(* IEC 61131-3 sources: xPLCCore/codesys_code/Application (part 2) *)

(* ---- PRG_DiagReply.st ---- *)
PROGRAM PRG_DiagReply
VAR_INPUT
    // Request: one SYS packet copied in by TCP_MSGPAK_Server (Comm task),
    // ReqLen > 0 means "answer it this call"; cleared when done. Inputs,
    // so the caller may write them.
    ReqBuf  : ARRAY[0..255] OF BYTE;
    ReqLen  : UDINT;
END_VAR
VAR
    // Reply, ready for fbMyServer.Send when OutLen > 0 (one call = one reply).
    OutBuf  : ARRAY[0..2047] OF BYTE;
    OutLen  : UDINT;
    DiagInfo  : MsgPakInfo;
    xInfoInit : BOOL;

    // Same names as in AxisGroupSM so the handler code moved here on
    // 2026-10-05 reads unchanged (own instances: this is another task).
    MessagePackerFb       : FB_MpPacker;
    MessageUnpackerFb     : FB_MpUnpacker;
    ResponsePacketPointer : POINTER TO MsgPakInfo;
    CommandId   : DINT;
    CommandType : STRING;
    CommandAck  : BOOL;
    ShouldReturn : BOOL;

    HandledCount : UDINT;     // replies built
    UnknownCount : UDINT;     // a command routed here without a handler

    // Scratch (was AxisGroupSM.DrainHostPackets VAR).
    EcTrStr : STRING(255);    // EC_STATS trl / trh
    EcSnapK : INT;
    EcObjJ  : INT;
    EcObjKey : STRING(7);
    EcTrI   : INT;
    EcEvtFrom : UDINT;
    EcEvtI  : UDINT;
    // TASK_STATS scratch.
    TsH     : __XWORD;        // RTS_IEC_HANDLE
    TsR     : UDINT;          // RTS_IEC_RESULT, 0 = ERR_OK
    TsP     : POINTER TO CmpIecTask.Task_Info2;
    TsN     : INT;
    TsReset : BOOL;
    TsKey   : STRING(31);
    TsName  : STRING(63);
END_VAR
(* =========== IMPLEMENTATION =========== *)
// Read-only diagnostics answered in the Comm task (2026-10-05). These
// commands only read GVL / AxisGroupSM state (a few set a reset flag that
// the EtherCAT task consumes), and their replies are long (EC_STATS ~1 KB,
// TASK_STATS, DEM_STATS snap): built in the 1 ms EtherCAT task they could
// make a scan overrun. TCP_MSGPAK_Server copies the packet into ReqBuf and
// calls this program, then sends OutBuf itself, so the reply ring
// (reMP_info) keeps its single producer. Not in a task of its own.
//
// The handler bodies are the ones that lived in AxisGroupSM.DrainHostPackets;
// AxisGroupSM.* reads are a torn-read risk only in theory (diagnostics).
OutLen := 0;
IF ReqLen = 0 THEN
    RETURN;
END_IF;
IF NOT xInfoInit THEN
    DiagInfo := MsgPakInfoInit(ADR(OutBuf), 2048, TRUE);
    xInfoInit := TRUE;
END_IF;
MsgPakInfoClear(DiagInfo);
ResponsePacketPointer := ADR(DiagInfo);
MessagePackerFb.BindSlot(ResponsePacketPointer);
MessageUnpackerFb.Init(ADR(ReqBuf), ReqLen);
CommandId   := TO_DINT(MessageUnpackerFb.TryReadINT64('id', 0));
CommandType := MessageUnpackerFb.TryReadString('cmd', '');
CommandAck  := FALSE;
ShouldReturn := FALSE;

    IF (CommandType = 'SETTLE_TRACE') THEN
        // The last stop trace (GVL.Tr*): seq, at (PLC ms of the stop),
        // ev = up to 4 samples from index from:i (0..399, 100 = the
        // stop) as cx:cy:cz:ax:ay:az (mm), comma separated.
        ShouldReturn := TRUE;
        CommandAck := TRUE;
        ResponsePacketPointer^.ele_count := 0;
        EcTrI := LIMIT(0, LINT_TO_INT(MessageUnpackerFb.TryReadINT64('from', 0)), 399);
        MessagePackerFb.PackKvLint(ADR('seq'), UDINT_TO_LINT(GVL.TrSeq));
        MessagePackerFb.PackKvLint(ADR('at'), UDINT_TO_LINT(GVL.TrAtMs));
        EcTrStr := '';
        FOR EcObjJ := EcTrI TO MIN(EcTrI + 3, 399) DO
            EcTrStr := CONCAT(EcTrStr, REAL_TO_STRING(GVL.TrCX[EcObjJ]));
            EcTrStr := CONCAT(EcTrStr, ':');
            EcTrStr := CONCAT(EcTrStr, REAL_TO_STRING(GVL.TrCY[EcObjJ]));
            EcTrStr := CONCAT(EcTrStr, ':');
            EcTrStr := CONCAT(EcTrStr, REAL_TO_STRING(GVL.TrCZ[EcObjJ]));
            EcTrStr := CONCAT(EcTrStr, ':');
            EcTrStr := CONCAT(EcTrStr, REAL_TO_STRING(GVL.TrAX[EcObjJ]));
            EcTrStr := CONCAT(EcTrStr, ':');
            EcTrStr := CONCAT(EcTrStr, REAL_TO_STRING(GVL.TrAY[EcObjJ]));
            EcTrStr := CONCAT(EcTrStr, ':');
            EcTrStr := CONCAT(EcTrStr, REAL_TO_STRING(GVL.TrAZ[EcObjJ]));
            EcTrStr := CONCAT(EcTrStr, ',');
        END_FOR;
        MessagePackerFb.PackKvStr(ADR('ev'), ADR(EcTrStr));
    ELSIF (CommandType = 'SETTLE') THEN
        // Settling-time log (GVL.Settle*): n = stops so far, tol =
        // tolerance mm, ev = up to 20 stops from index from:i as
        // at_ms:settle_ms:err_at_stop_um. reset:1 clears it.
        ShouldReturn := TRUE;
        CommandAck := TRUE;
        ResponsePacketPointer^.ele_count := 0;
        IF MessageUnpackerFb.TryReadINT64('reset', 0) <> 0 THEN
            GVL.SettleN := 0;
        END_IF;
        EcEvtFrom := LINT_TO_UDINT(MessageUnpackerFb.TryReadINT64('from', 0));
        MessagePackerFb.PackKvLint(ADR('n'), UDINT_TO_LINT(GVL.SettleN));
        MessagePackerFb.PackKvReal(ADR('tol'), LREAL_TO_REAL(GVL.SettleTolMm));
        EcTrStr := '';
        EcEvtI := EcEvtFrom;
        WHILE (EcEvtI < GVL.SettleN) AND (EcEvtI < EcEvtFrom + 20) DO
            EcTrStr := CONCAT(EcTrStr, UDINT_TO_STRING(GVL.SettleAtMs[EcEvtI MOD 256]));
            EcTrStr := CONCAT(EcTrStr, ':');
            EcTrStr := CONCAT(EcTrStr, UDINT_TO_STRING(GVL.SettleMs[EcEvtI MOD 256]));
            EcTrStr := CONCAT(EcTrStr, ':');
            EcTrStr := CONCAT(EcTrStr, UDINT_TO_STRING(GVL.SettleErrUm[EcEvtI MOD 256]));
            EcTrStr := CONCAT(EcTrStr, ',');
            EcEvtI := EcEvtI + 1;
        END_WHILE;
        MessagePackerFb.PackKvStr(ADR('ev'), ADR(EcTrStr));
    ELSIF (CommandType = 'DWELL') THEN
        // Every-stop log (GVL.Dw*): n = stops so far, tol mm, hist =
        // settle time histogram (edges 1 2 5 10 15 20 50 ms, last =
        // not settled), emax = max error when leaving (um), ev = up
        // to 8 stops from index from:i as at_ms:dwell_ms:settle_ms:
        // err_stop_um:err_leave_um:err_5ms_um:err_10ms_um (settle 4294967295
        // = not settled; fields 6 and 7 since 2026-10-05); evq = the same
        // stops as buf:hostq:cool_ms:z_um (GVL.DwBuf / DwHostQ / DwCoolMs /
        // DwZUm, 2026-10-05; a separate string so ev stays within 255).
        // reset:1 clears it.
        ShouldReturn := TRUE;
        CommandAck := TRUE;
        ResponsePacketPointer^.ele_count := 0;
        IF MessageUnpackerFb.TryReadINT64('reset', 0) <> 0 THEN
            GVL.DwN := 0;
            GVL.DwErrLeaveMaxUm := 0;
            FOR EcObjJ := 0 TO 8 DO
                GVL.DwHist[EcObjJ] := 0;
            END_FOR;
        END_IF;
        EcEvtFrom := LINT_TO_UDINT(MessageUnpackerFb.TryReadINT64('from', 0));
        MessagePackerFb.PackKvLint(ADR('n'), UDINT_TO_LINT(GVL.DwN));
        MessagePackerFb.PackKvReal(ADR('tol'), LREAL_TO_REAL(GVL.SettleTolMm));
        MessagePackerFb.PackKvLint(ADR('emax'), UDINT_TO_LINT(GVL.DwErrLeaveMaxUm));
        EcTrStr := '';
        FOR EcObjJ := 0 TO 8 DO
            EcTrStr := CONCAT(EcTrStr, UDINT_TO_STRING(GVL.DwHist[EcObjJ]));
            EcTrStr := CONCAT(EcTrStr, ',');
        END_FOR;
        MessagePackerFb.PackKvStr(ADR('hist'), ADR(EcTrStr));
        EcTrStr := '';
        EcEvtI := EcEvtFrom;
        WHILE (EcEvtI < GVL.DwN) AND (EcEvtI < EcEvtFrom + 8) DO
            EcTrStr := CONCAT(EcTrStr, UDINT_TO_STRING(GVL.DwAtMs[EcEvtI MOD 4096]));
            EcTrStr := CONCAT(EcTrStr, ':');
            EcTrStr := CONCAT(EcTrStr, UDINT_TO_STRING(GVL.DwDwellMs[EcEvtI MOD 4096]));
            EcTrStr := CONCAT(EcTrStr, ':');
            EcTrStr := CONCAT(EcTrStr, UDINT_TO_STRING(GVL.DwSettleMs[EcEvtI MOD 4096]));
            EcTrStr := CONCAT(EcTrStr, ':');
            EcTrStr := CONCAT(EcTrStr, UDINT_TO_STRING(GVL.DwErr0Um[EcEvtI MOD 4096]));
            EcTrStr := CONCAT(EcTrStr, ':');
            EcTrStr := CONCAT(EcTrStr, UDINT_TO_STRING(GVL.DwErrLeaveUm[EcEvtI MOD 4096]));
            EcTrStr := CONCAT(EcTrStr, ':');
            EcTrStr := CONCAT(EcTrStr, UDINT_TO_STRING(GVL.DwErr5Um[EcEvtI MOD 4096]));
            EcTrStr := CONCAT(EcTrStr, ':');
            EcTrStr := CONCAT(EcTrStr, UDINT_TO_STRING(GVL.DwErr10Um[EcEvtI MOD 4096]));
            EcTrStr := CONCAT(EcTrStr, ',');
            EcEvtI := EcEvtI + 1;
        END_WHILE;
        MessagePackerFb.PackKvStr(ADR('ev'), ADR(EcTrStr));
        EcTrStr := '';
        EcEvtI := EcEvtFrom;
        WHILE (EcEvtI < GVL.DwN) AND (EcEvtI < EcEvtFrom + 8) DO
            EcTrStr := CONCAT(EcTrStr, UINT_TO_STRING(GVL.DwBuf[EcEvtI MOD 4096]));
            EcTrStr := CONCAT(EcTrStr, ':');
            EcTrStr := CONCAT(EcTrStr, UINT_TO_STRING(GVL.DwHostQ[EcEvtI MOD 4096]));
            EcTrStr := CONCAT(EcTrStr, ':');
            EcTrStr := CONCAT(EcTrStr, INT_TO_STRING(GVL.DwCoolMs[EcEvtI MOD 4096]));
            EcTrStr := CONCAT(EcTrStr, ':');
            EcTrStr := CONCAT(EcTrStr, DINT_TO_STRING(GVL.DwZUm[EcEvtI MOD 4096]));
            EcTrStr := CONCAT(EcTrStr, ',');
            EcEvtI := EcEvtI + 1;
        END_WHILE;
        MessagePackerFb.PackKvStr(ADR('evq'), ADR(EcTrStr));
    ELSIF (CommandType = 'FB_STATS') THEN
        // Feedback shock monitor (GVL.Fb*): per drive k, fd{k} =
        // histogram of |d2 actual position| (edges 1k 2k 5k 10k 20k
        // 50k 100k PUU), fdm{k} its max, ft{k} = histogram of |torque
        // change| (edges 5 10 20 50 100 200 500, 0.1 %), ftm{k} its
        // max, tq{k} = the torque now. reset:1 clears after the reply.
        ShouldReturn := TRUE;
        CommandAck := TRUE;
        ResponsePacketPointer^.ele_count := 0;
        FOR EcTrI := 0 TO 2 DO
            EcTrStr := '';
            FOR EcObjJ := 0 TO 7 DO
                EcTrStr := CONCAT(EcTrStr, UDINT_TO_STRING(GVL.FbD2Hist[EcTrI, EcObjJ]));
                EcTrStr := CONCAT(EcTrStr, ',');
            END_FOR;
            EcObjKey := CONCAT('fd', INT_TO_STRING(EcTrI));
            MessagePackerFb.PackKvStr(ADR(EcObjKey), ADR(EcTrStr));
            EcObjKey := CONCAT('fdm', INT_TO_STRING(EcTrI));
            MessagePackerFb.PackKvDint(ADR(EcObjKey), GVL.FbD2Max[EcTrI]);
            EcTrStr := '';
            FOR EcObjJ := 0 TO 7 DO
                EcTrStr := CONCAT(EcTrStr, UDINT_TO_STRING(GVL.FbTqHist[EcTrI, EcObjJ]));
                EcTrStr := CONCAT(EcTrStr, ',');
            END_FOR;
            EcObjKey := CONCAT('ft', INT_TO_STRING(EcTrI));
            MessagePackerFb.PackKvStr(ADR(EcObjKey), ADR(EcTrStr));
            EcObjKey := CONCAT('ftm', INT_TO_STRING(EcTrI));
            MessagePackerFb.PackKvDint(ADR(EcObjKey), INT_TO_DINT(GVL.FbTqMax[EcTrI]));
        END_FOR;
        MessagePackerFb.PackKvDint(ADR('tq0'), INT_TO_DINT(GVL.TorqueTap0));
        MessagePackerFb.PackKvDint(ADR('tq1'), INT_TO_DINT(GVL.TorqueTap1));
        MessagePackerFb.PackKvDint(ADR('tq2'), INT_TO_DINT(GVL.TorqueTap2));
        IF MessageUnpackerFb.TryReadINT64('reset', 0) <> 0 THEN
            GVL.FbReset := TRUE;
        END_IF;
    ELSIF (CommandType = 'ESP_SYNC') THEN
        // The EasyCAT SYNC0-interval log (GVL.SyncLog*): n = buckets
        // so far, now = the last deviation (ns), ev = up to 12
        // buckets from index from:i as ms:min:max (ns).
        ShouldReturn := TRUE;
        CommandAck := TRUE;
        ResponsePacketPointer^.ele_count := 0;
        EcEvtFrom := LINT_TO_UDINT(MessageUnpackerFb.TryReadINT64('from', 0));
        MessagePackerFb.PackKvLint(ADR('n'), UDINT_TO_LINT(GVL.SyncLogN));
        MessagePackerFb.PackKvDint(ADR('now'), INT_TO_DINT(GVL.EspSyncDevNs));
        EcTrStr := '';
        EcEvtI := EcEvtFrom;
        WHILE (EcEvtI < GVL.SyncLogN) AND (EcEvtI < EcEvtFrom + 12) DO
            EcTrStr := CONCAT(EcTrStr, UDINT_TO_STRING(GVL.SyncLogMs[EcEvtI MOD 4096]));
            EcTrStr := CONCAT(EcTrStr, ':');
            EcTrStr := CONCAT(EcTrStr, INT_TO_STRING(GVL.SyncLogMin[EcEvtI MOD 4096]));
            EcTrStr := CONCAT(EcTrStr, ':');
            EcTrStr := CONCAT(EcTrStr, INT_TO_STRING(GVL.SyncLogMax[EcEvtI MOD 4096]));
            EcTrStr := CONCAT(EcTrStr, ',');
            EcEvtI := EcEvtI + 1;
        END_WHILE;
        MessagePackerFb.PackKvStr(ADR('ev'), ADR(EcTrStr));
    ELSIF (CommandType = 'ESP_ARR') THEN
        // The EasyCAT frame-arrival log (GVL.ArrLog*): n = buckets so
        // far, now = the last arrival (us), ev = up to 12 buckets from
        // index from:i as ms:min:max (us), comma separated.
        ShouldReturn := TRUE;
        CommandAck := TRUE;
        ResponsePacketPointer^.ele_count := 0;
        EcEvtFrom := LINT_TO_UDINT(MessageUnpackerFb.TryReadINT64('from', 0));
        MessagePackerFb.PackKvLint(ADR('n'), UDINT_TO_LINT(GVL.ArrLogN));
        MessagePackerFb.PackKvDint(ADR('now'), UINT_TO_DINT(GVL.EspArrUs));
        EcTrStr := '';
        EcEvtI := EcEvtFrom;
        WHILE (EcEvtI < GVL.ArrLogN) AND (EcEvtI < EcEvtFrom + 12) DO
            EcTrStr := CONCAT(EcTrStr, UDINT_TO_STRING(GVL.ArrLogMs[EcEvtI MOD 4096]));
            EcTrStr := CONCAT(EcTrStr, ':');
            EcTrStr := CONCAT(EcTrStr, UINT_TO_STRING(GVL.ArrLogMin[EcEvtI MOD 4096]));
            EcTrStr := CONCAT(EcTrStr, ':');
            EcTrStr := CONCAT(EcTrStr, UINT_TO_STRING(GVL.ArrLogMax[EcEvtI MOD 4096]));
            EcTrStr := CONCAT(EcTrStr, ',');
            EcEvtI := EcEvtI + 1;
        END_WHILE;
        MessagePackerFb.PackKvStr(ADR('ev'), ADR(EcTrStr));
    ELSIF (CommandType = 'DEM_EVT') THEN
        // The delay-change event log of drive axis:k (GVL.DemEvt):
        // n = events so far, ev = up to 20 entries from index from:i
        // (ms * 4 + code, comma separated). Entries older than
        // n - 1024 are overwritten.
        ShouldReturn := TRUE;
        CommandAck := TRUE;
        ResponsePacketPointer^.ele_count := 0;
        EcTrI := LIMIT(0, LINT_TO_INT(MessageUnpackerFb.TryReadINT64('axis', 0)), 2);
        EcEvtFrom := LINT_TO_UDINT(MessageUnpackerFb.TryReadINT64('from', 0));
        MessagePackerFb.PackKvLint(ADR('n'), UDINT_TO_LINT(GVL.DemEvtN[EcTrI]));
        EcTrStr := '';
        EcEvtI := EcEvtFrom;
        WHILE (EcEvtI < GVL.DemEvtN[EcTrI]) AND (EcEvtI < EcEvtFrom + 20) DO
            EcTrStr := CONCAT(EcTrStr, UDINT_TO_STRING(GVL.DemEvt[EcTrI, EcEvtI MOD 1024]));
            EcTrStr := CONCAT(EcTrStr, ',');
            EcEvtI := EcEvtI + 1;
        END_WHILE;
        MessagePackerFb.PackKvStr(ADR('ev'), ADR(EcTrStr));
    ELSIF (CommandType = 'DEM_STATS') THEN
        // The drives' position demand (0x6062) vs the targets we sent
        // (GVL.Dem*, PRG_EventLog). Per drive k: ds{k} stale, dlate{k}
        // one cycle behind the nominal lag, dgl{k} / dmx{k} d2 glitches /
        // max, dlt{k} PLC ms of the last stale, dl{k} the lag histogram
        // as text (lag 0..6, none). nsnap = snapshots taken; snap:i adds
        // snapshot i (s_axis, s_ms, s_why, s_t0 / s_t1 and s_d0 / s_d1 =
        // cycles 0-15 / 16-31 of target / demand). reset:1 clears.
        ShouldReturn := TRUE;
        CommandAck := TRUE;
        ResponsePacketPointer^.ele_count := 0;
        MessagePackerFb.PackKvDint(ADR('lagnom'), INT_TO_DINT(GVL.DemLagNominal));
        FOR EcTrI := 0 TO 2 DO
            EcObjKey := CONCAT('ds', INT_TO_STRING(EcTrI));
            MessagePackerFb.PackKvLint(ADR(EcObjKey), UDINT_TO_LINT(GVL.DemStale[EcTrI]));
            EcObjKey := CONCAT('dlate', INT_TO_STRING(EcTrI));
            MessagePackerFb.PackKvLint(ADR(EcObjKey), UDINT_TO_LINT(GVL.DemLate[EcTrI]));
            EcObjKey := CONCAT('dgl', INT_TO_STRING(EcTrI));
            MessagePackerFb.PackKvLint(ADR(EcObjKey), UDINT_TO_LINT(GVL.DemGlitch[EcTrI]));
            EcObjKey := CONCAT('dmx', INT_TO_STRING(EcTrI));
            MessagePackerFb.PackKvDint(ADR(EcObjKey), GVL.DemD2Max[EcTrI]);
            EcObjKey := CONCAT('dlt', INT_TO_STRING(EcTrI));
            MessagePackerFb.PackKvLint(ADR(EcObjKey), UDINT_TO_LINT(GVL.DemLastStaleMs[EcTrI]));
            EcTrStr := '';
            FOR EcObjJ := 0 TO 7 DO
                EcTrStr := CONCAT(EcTrStr, UDINT_TO_STRING(GVL.DemLag[EcTrI, EcObjJ]));
                EcTrStr := CONCAT(EcTrStr, ',');
            END_FOR;
            EcObjKey := CONCAT('dl', INT_TO_STRING(EcTrI));
            MessagePackerFb.PackKvStr(ADR(EcObjKey), ADR(EcTrStr));
        END_FOR;
        FOR EcTrI := 0 TO 2 DO
            EcObjKey := CONCAT('soff', INT_TO_STRING(EcTrI));
            MessagePackerFb.PackKvLint(ADR(EcObjKey), UDINT_TO_LINT(GVL.SyncOffCount[EcTrI]));
            EcObjKey := CONCAT('sofl', INT_TO_STRING(EcTrI));
            MessagePackerFb.PackKvLint(ADR(EcObjKey), UDINT_TO_LINT(GVL.SyncOffAndLate[EcTrI]));
            EcObjKey := CONCAT('stat', INT_TO_STRING(EcTrI));
            CASE EcTrI OF
                0: MessagePackerFb.PackKvDint(ADR(EcObjKey), WORD_TO_DINT(GVL.StatusTap0));
                1: MessagePackerFb.PackKvDint(ADR(EcObjKey), WORD_TO_DINT(GVL.StatusTap1));
            ELSE
                MessagePackerFb.PackKvDint(ADR(EcObjKey), WORD_TO_DINT(GVL.StatusTap2));
            END_CASE;
        END_FOR;
        MessagePackerFb.PackKvDint(ADR('nsnap'), INT_TO_DINT(GVL.DemSnapN));
        EcTrI := LINT_TO_INT(MessageUnpackerFb.TryReadINT64('snap', -1));
        IF (EcTrI >= 0) AND (EcTrI < GVL.DemSnapN) THEN
            MessagePackerFb.PackKvDint(ADR('s_axis'), INT_TO_DINT(GVL.DemSnapAxis[EcTrI]));
            MessagePackerFb.PackKvLint(ADR('s_ms'), UDINT_TO_LINT(GVL.DemSnapMs[EcTrI]));
            MessagePackerFb.PackKvDint(ADR('s_why'), INT_TO_DINT(GVL.DemSnapWhy[EcTrI]));
            EcTrStr := '';
            FOR EcSnapK := 0 TO 31 DO
                IF (GVL.DemSnapS[EcTrI, EcSnapK] AND 16#4000) <> 0 THEN
                    EcTrStr := CONCAT(EcTrStr, '1');
                ELSE
                    EcTrStr := CONCAT(EcTrStr, '0');
                END_IF;
            END_FOR;
            MessagePackerFb.PackKvStr(ADR('s_sync'), ADR(EcTrStr));
            FOR EcObjJ := 0 TO 3 DO
                EcTrStr := '';
                FOR EcSnapK := 0 TO 15 DO
                    IF EcObjJ < 2 THEN
                        EcTrStr := CONCAT(EcTrStr, DINT_TO_STRING(GVL.DemSnapT[EcTrI, (EcObjJ MOD 2) * 16 + EcSnapK]));
                    ELSE
                        EcTrStr := CONCAT(EcTrStr, DINT_TO_STRING(GVL.DemSnapD[EcTrI, (EcObjJ MOD 2) * 16 + EcSnapK]));
                    END_IF;
                    EcTrStr := CONCAT(EcTrStr, ',');
                END_FOR;
                CASE EcObjJ OF
                    0: EcObjKey := 's_t0';
                    1: EcObjKey := 's_t1';
                    2: EcObjKey := 's_d0';
                ELSE
                    EcObjKey := 's_d1';
                END_CASE;
                MessagePackerFb.PackKvStr(ADR(EcObjKey), ADR(EcTrStr));
            END_FOR;
        END_IF;
        IF MessageUnpackerFb.TryReadINT64('reset', 0) <> 0 THEN
            GVL.DemReset := TRUE;
        END_IF;
    ELSIF (CommandType = 'EC_STATS') THEN
        // EtherCAT health: the master's frame statistics (lost /
        // tx_err / rx_err, updated every 100 cycles) and the task
        // timing monitor (GVL.EcProf*: cycles, late100 / late500 =
        // periods over nominal + 100 / 500 us, pmin / pmax us,
        // h0..h5 = |period - nominal| < 20/50/100/200/500/>=500 us,
        // dc_out = cycles with DC out of sync, agsm_max us). reset:1
        // starts all of them over after this reply.
        ShouldReturn := TRUE;
        CommandAck := TRUE;
        ResponsePacketPointer^.ele_count := 0;
        MessagePackerFb.PackKvLint(ADR('lost'), UDINT_TO_LINT(GVL.EcLostFrames));
        MessagePackerFb.PackKvLint(ADR('tx_err'), UDINT_TO_LINT(GVL.EcTxErrors));
        MessagePackerFb.PackKvLint(ADR('rx_err'), UDINT_TO_LINT(GVL.EcRxErrors));
        MessagePackerFb.PackKvLint(ADR('cycles'), UDINT_TO_LINT(GVL.EcProfCycles));
        MessagePackerFb.PackKvLint(ADR('late100'), UDINT_TO_LINT(GVL.EcLate100));
        MessagePackerFb.PackKvLint(ADR('late500'), UDINT_TO_LINT(GVL.EcLate500));
        MessagePackerFb.PackKvReal(ADR('pmin'), LREAL_TO_REAL(GVL.EcPeriodUsMin));
        MessagePackerFb.PackKvReal(ADR('pmax'), LREAL_TO_REAL(GVL.EcPeriodUsMax));
        MessagePackerFb.PackKvLint(ADR('h0'), UDINT_TO_LINT(GVL.EcPeriodHist[0]));
        MessagePackerFb.PackKvLint(ADR('h1'), UDINT_TO_LINT(GVL.EcPeriodHist[1]));
        MessagePackerFb.PackKvLint(ADR('h2'), UDINT_TO_LINT(GVL.EcPeriodHist[2]));
        MessagePackerFb.PackKvLint(ADR('h3'), UDINT_TO_LINT(GVL.EcPeriodHist[3]));
        MessagePackerFb.PackKvLint(ADR('h4'), UDINT_TO_LINT(GVL.EcPeriodHist[4]));
        MessagePackerFb.PackKvLint(ADR('h5'), UDINT_TO_LINT(GVL.EcPeriodHist[5]));
        MessagePackerFb.PackKvLint(ADR('dc_out'), UDINT_TO_LINT(GVL.EcDcOutCycles));
        MessagePackerFb.PackKvReal(ADR('agsm_max'), LREAL_TO_REAL(GVL.EcAgsmUsMax));
        // g0..2 / gms0..2 / d2m0..2: set-position glitches of the
        // delta joints (count, PLC ms of the last, max |d2| deg/cycle^2)
        MessagePackerFb.PackKvLint(ADR('g0'), UDINT_TO_LINT(GVL.SetGlitchCount[0]));
        MessagePackerFb.PackKvLint(ADR('g1'), UDINT_TO_LINT(GVL.SetGlitchCount[1]));
        MessagePackerFb.PackKvLint(ADR('g2'), UDINT_TO_LINT(GVL.SetGlitchCount[2]));
        MessagePackerFb.PackKvLint(ADR('gms0'), UDINT_TO_LINT(GVL.SetGlitchLastMs[0]));
        MessagePackerFb.PackKvLint(ADR('gms1'), UDINT_TO_LINT(GVL.SetGlitchLastMs[1]));
        MessagePackerFb.PackKvLint(ADR('gms2'), UDINT_TO_LINT(GVL.SetGlitchLastMs[2]));
        MessagePackerFb.PackKvReal(ADR('d2m0'), LREAL_TO_REAL(GVL.SetD2Max[0]));
        MessagePackerFb.PackKvReal(ADR('d2m1'), LREAL_TO_REAL(GVL.SetD2Max[1]));
        MessagePackerFb.PackKvReal(ADR('d2m2'), LREAL_TO_REAL(GVL.SetD2Max[2]));
        // tic_max / tic0..9: where the task's IEC code ends in the
        // DC cycle (us, 100 us bins); sm0..2 / se0..2: the drives'
        // 0x1C32:0B SM-event missed / :20 sync error (-1 = SDO
        // failed, sdo_err)
        MessagePackerFb.PackKvReal(ADR('tic_max'), LREAL_TO_REAL(GVL.EcTicUsMax));
        MessagePackerFb.PackKvLint(ADR('tic0'), UDINT_TO_LINT(GVL.EcTicHist[0]));
        MessagePackerFb.PackKvLint(ADR('tic1'), UDINT_TO_LINT(GVL.EcTicHist[1]));
        MessagePackerFb.PackKvLint(ADR('tic2'), UDINT_TO_LINT(GVL.EcTicHist[2]));
        MessagePackerFb.PackKvLint(ADR('tic3'), UDINT_TO_LINT(GVL.EcTicHist[3]));
        MessagePackerFb.PackKvLint(ADR('tic4'), UDINT_TO_LINT(GVL.EcTicHist[4]));
        MessagePackerFb.PackKvLint(ADR('tic5'), UDINT_TO_LINT(GVL.EcTicHist[5]));
        MessagePackerFb.PackKvLint(ADR('tic6'), UDINT_TO_LINT(GVL.EcTicHist[6]));
        MessagePackerFb.PackKvLint(ADR('tic7'), UDINT_TO_LINT(GVL.EcTicHist[7]));
        MessagePackerFb.PackKvLint(ADR('tic8'), UDINT_TO_LINT(GVL.EcTicHist[8]));
        MessagePackerFb.PackKvLint(ADR('tic9'), UDINT_TO_LINT(GVL.EcTicHist[9]));
        MessagePackerFb.PackKvDint(ADR('sm0'), GVL.DrvSmMissed[0]);
        MessagePackerFb.PackKvDint(ADR('sm1'), GVL.DrvSmMissed[1]);
        MessagePackerFb.PackKvDint(ADR('sm2'), GVL.DrvSmMissed[2]);
        MessagePackerFb.PackKvDint(ADR('se0'), GVL.DrvSyncErr[0]);
        MessagePackerFb.PackKvDint(ADR('se1'), GVL.DrvSyncErr[1]);
        MessagePackerFb.PackKvDint(ADR('se2'), GVL.DrvSyncErr[2]);
        MessagePackerFb.PackKvDint(ADR('sdo_err'), GVL.EcSdoErr);
        MessagePackerFb.PackKvLint(ADR('bus_us'), DWORD_TO_LINT(AxisGroupSM.BusPeriodUs));   // EtherCAT_Task interval as read
        // Comm task profile: cs0..2 worst segment us (TCP server / MbProbe / EspHttp),
        // cb0..2 bus cycles inside it, co0..2 segments > 1 ms, cscan worst whole scan
        MessagePackerFb.PackKvReal(ADR('cs0'), LREAL_TO_REAL(GVL.CommSegUsMax[0]));
        MessagePackerFb.PackKvLint(ADR('cb0'), UDINT_TO_LINT(GVL.CommSegBusCyc[0]));
        MessagePackerFb.PackKvLint(ADR('co0'), UDINT_TO_LINT(GVL.CommSegOver1ms[0]));
        MessagePackerFb.PackKvReal(ADR('cs1'), LREAL_TO_REAL(GVL.CommSegUsMax[1]));
        MessagePackerFb.PackKvLint(ADR('cb1'), UDINT_TO_LINT(GVL.CommSegBusCyc[1]));
        MessagePackerFb.PackKvLint(ADR('co1'), UDINT_TO_LINT(GVL.CommSegOver1ms[1]));
        MessagePackerFb.PackKvReal(ADR('cs2'), LREAL_TO_REAL(GVL.CommSegUsMax[2]));
        MessagePackerFb.PackKvLint(ADR('cb2'), UDINT_TO_LINT(GVL.CommSegBusCyc[2]));
        MessagePackerFb.PackKvLint(ADR('co2'), UDINT_TO_LINT(GVL.CommSegOver1ms[2]));
        MessagePackerFb.PackKvReal(ADR('cscan'), LREAL_TO_REAL(GVL.CommScanUsMax));
        // fj0..3 / fm0..3 / fl0..3: following-error jumps (EAxis0..2, reel): count, max, PLC ms of the last
        MessagePackerFb.PackKvLint(ADR('fj0'), UDINT_TO_LINT(GVL.FeJumpCount[0]));
        MessagePackerFb.PackKvReal(ADR('fm0'), LREAL_TO_REAL(GVL.FeJumpMax[0]));
        MessagePackerFb.PackKvLint(ADR('fl0'), UDINT_TO_LINT(GVL.FeLastJumpMs[0]));
        MessagePackerFb.PackKvLint(ADR('fj1'), UDINT_TO_LINT(GVL.FeJumpCount[1]));
        MessagePackerFb.PackKvReal(ADR('fm1'), LREAL_TO_REAL(GVL.FeJumpMax[1]));
        MessagePackerFb.PackKvLint(ADR('fl1'), UDINT_TO_LINT(GVL.FeLastJumpMs[1]));
        MessagePackerFb.PackKvLint(ADR('fj2'), UDINT_TO_LINT(GVL.FeJumpCount[2]));
        MessagePackerFb.PackKvReal(ADR('fm2'), LREAL_TO_REAL(GVL.FeJumpMax[2]));
        MessagePackerFb.PackKvLint(ADR('fl2'), UDINT_TO_LINT(GVL.FeLastJumpMs[2]));
        MessagePackerFb.PackKvLint(ADR('fj3'), UDINT_TO_LINT(GVL.FeJumpCount[3]));
        MessagePackerFb.PackKvReal(ADR('fm3'), LREAL_TO_REAL(GVL.FeJumpMax[3]));
        MessagePackerFb.PackKvLint(ADR('fl3'), UDINT_TO_LINT(GVL.FeLastJumpMs[3]));
        MessagePackerFb.PackKvReal(ADR('ctask'), LREAL_TO_REAL(GVL.CommTaskUsMax));
        MessagePackerFb.PackKvReal(ADR('cout'), LREAL_TO_REAL(GVL.CommOutsideUsMax));
        MessagePackerFb.PackKvLint(ADR('cout500'), UDINT_TO_LINT(GVL.CommOutsideOver500));
        IF MessageUnpackerFb.TryReadINT64('obj', 0) <> 0 THEN  // long text: only on request
            // o0..o2: drive k's sync objects (DrvObj), "v,v,..." text
            FOR EcTrI := 0 TO 2 DO
                EcTrStr := '';
                FOR EcObjJ := 0 TO 11 DO
                    EcTrStr := CONCAT(EcTrStr, DINT_TO_STRING(GVL.DrvObj[EcTrI, EcObjJ]));
                    EcTrStr := CONCAT(EcTrStr, ',');
                END_FOR;
                EcObjKey := CONCAT('o', INT_TO_STRING(EcTrI));
                MessagePackerFb.PackKvStr(ADR(EcObjKey), ADR(EcTrStr));
            END_FOR;
        END_IF;
        // dg0..2 / dd0..2: the same glitch check on the integer
        // target sent to the drive (diSetPosition): count, max |d2|
        MessagePackerFb.PackKvLint(ADR('dg0'), UDINT_TO_LINT(GVL.DiGlitchCount[0]));
        MessagePackerFb.PackKvLint(ADR('dg1'), UDINT_TO_LINT(GVL.DiGlitchCount[1]));
        MessagePackerFb.PackKvLint(ADR('dg2'), UDINT_TO_LINT(GVL.DiGlitchCount[2]));
        MessagePackerFb.PackKvDint(ADR('dd0'), GVL.DiD2Max[0]);
        MessagePackerFb.PackKvDint(ADR('dd1'), GVL.DiD2Max[1]);
        MessagePackerFb.PackKvDint(ADR('dd2'), GVL.DiD2Max[2]);
        // tap*: the Target Position in the output image (read-only AT taps)
        MessagePackerFb.PackKvLint(ADR('tg0'), UDINT_TO_LINT(GVL.TapGlitch[0]));
        MessagePackerFb.PackKvDint(ADR('td0'), GVL.TapD2Max[0]);
        MessagePackerFb.PackKvLint(ADR('tnow0'), UDINT_TO_LINT(GVL.TapEqNow[0]));
        MessagePackerFb.PackKvLint(ADR('tprev0'), UDINT_TO_LINT(GVL.TapEqPrev[0]));
        MessagePackerFb.PackKvLint(ADR('tnone0'), UDINT_TO_LINT(GVL.TapEqNone[0]));
        MessagePackerFb.PackKvLint(ADR('tg1'), UDINT_TO_LINT(GVL.TapGlitch[1]));
        MessagePackerFb.PackKvDint(ADR('td1'), GVL.TapD2Max[1]);
        MessagePackerFb.PackKvLint(ADR('tnow1'), UDINT_TO_LINT(GVL.TapEqNow[1]));
        MessagePackerFb.PackKvLint(ADR('tprev1'), UDINT_TO_LINT(GVL.TapEqPrev[1]));
        MessagePackerFb.PackKvLint(ADR('tnone1'), UDINT_TO_LINT(GVL.TapEqNone[1]));
        MessagePackerFb.PackKvLint(ADR('tg2'), UDINT_TO_LINT(GVL.TapGlitch[2]));
        MessagePackerFb.PackKvDint(ADR('td2'), GVL.TapD2Max[2]);
        MessagePackerFb.PackKvLint(ADR('tnow2'), UDINT_TO_LINT(GVL.TapEqNow[2]));
        MessagePackerFb.PackKvLint(ADR('tprev2'), UDINT_TO_LINT(GVL.TapEqPrev[2]));
        MessagePackerFb.PackKvLint(ADR('tnone2'), UDINT_TO_LINT(GVL.TapEqNone[2]));
        // EasyCAT bus timing probe: e_stale / e_skip since reset,
        // e_late last second, e_late_sum since reset (the arrival
        // min / max moved to the per-100-ms ArrLog, SYS ESP_ARR)
        MessagePackerFb.PackKvDint(ADR('e_stale'), UINT_TO_DINT(GVL.EspStale - GVL.EspStale0));
        MessagePackerFb.PackKvDint(ADR('e_skip'), UINT_TO_DINT(GVL.EspSkip - GVL.EspSkip0));
        MessagePackerFb.PackKvDint(ADR('e_late'), UINT_TO_DINT(GVL.EspLate));
        MessagePackerFb.PackKvLint(ADR('e_late_sum'), UDINT_TO_LINT(GVL.EspLateSum));
        // e_pg / e_pd2 / e_pd2peak: EAxis0's target stream checked on the ESP32
        MessagePackerFb.PackKvDint(ADR('e_pg'), UINT_TO_DINT(GVL.EspPosGlitch - GVL.EspPosGlitch0));
        MessagePackerFb.PackKvLint(ADR('e_pd2'), UDINT_TO_LINT(GVL.EspPosD2Max));
        MessagePackerFb.PackKvLint(ADR('e_pd2peak'), UDINT_TO_LINT(GVL.EspPosD2Peak));
        IF MessageUnpackerFb.TryReadINT64('tr', 0) <> 0 THEN   // long text: only on request
            // trl / trh: the last 20 x 500 ms min / max of the above,
            // oldest first ("lo0,..." as text, us)
            EcTrStr := '';
            FOR EcTrI := 0 TO 19 DO
                EcTrStr := CONCAT(EcTrStr, REAL_TO_STRING(GVL.EcTicTrMin[(GVL.EcTicIdx + EcTrI) MOD 20]));
                EcTrStr := CONCAT(EcTrStr, ',');
            END_FOR;
            MessagePackerFb.PackKvStr(ADR('trl'), ADR(EcTrStr));
            EcTrStr := '';
            FOR EcTrI := 0 TO 19 DO
                EcTrStr := CONCAT(EcTrStr, REAL_TO_STRING(GVL.EcTicTrMax[(GVL.EcTicIdx + EcTrI) MOD 20]));
                EcTrStr := CONCAT(EcTrStr, ',');
            END_FOR;
            MessagePackerFb.PackKvStr(ADR('trh'), ADR(EcTrStr));
        END_IF;
        IF MessageUnpackerFb.TryReadINT64('reset', 0) <> 0 THEN
            GVL.EcProfReset := TRUE;
            GVL.EcStatsClear := TRUE;
            GVL.CommProfReset := TRUE;
        END_IF;
    ELSIF (CommandType = 'TASK_STATS') THEN
        // The runtime's task statistics -- what the IDE's Task
        // Configuration > Monitor shows -- for every task of the
        // application, SoftMotion's planning task included. Flat
        // keys per task k: tk_name, tk_prio, tk_interval_us,
        // tk_last / tk_avg / tk_max / tk_min (cycle time, us),
        // tk_jit / tk_jmin / tk_jmax (jitter, us), tk_cycles,
        // tk_iec_cycles; n = tasks. reset:true zeroes them after
        // reading (as the IDE's reset does).
        ShouldReturn := TRUE;
        CommandAck := TRUE;
        ResponsePacketPointer^.ele_count := 0;
        TsReset := MessageUnpackerFb.TryReadINT64('reset', 0) <> 0;
        TsN := 0;
        TsH := CmpIecTask.IecTaskGetFirst(ADR('Application'), ADR(TsR));
        WHILE (TsR = 0) AND (TsN < 8) DO
            TsP := CmpIecTask.IecTaskGetInfo3(TsH, ADR(TsR));
            IF TsP <> 0 THEN
                IF TsP^.pszName <> 0 THEN
                    TsName := TsP^.pszName^;
                ELSE
                    TsName := '?';
                END_IF;
                TsKey := CONCAT(CONCAT('t', INT_TO_STRING(TsN)), '_name');
                MessagePackerFb.PackKvStr(ADR(TsKey), ADR(TsName));
                TsKey := CONCAT(CONCAT('t', INT_TO_STRING(TsN)), '_prio');
                MessagePackerFb.PackKvDint(ADR(TsKey), TsP^.nPriority);
                TsKey := CONCAT(CONCAT('t', INT_TO_STRING(TsN)), '_interval_us');
                MessagePackerFb.PackKvLint(ADR(TsKey), DWORD_TO_LINT(TsP^.dwInterval));
                TsKey := CONCAT(CONCAT('t', INT_TO_STRING(TsN)), '_last');
                MessagePackerFb.PackKvLint(ADR(TsKey), DWORD_TO_LINT(TsP^.dwCycleTime));
                TsKey := CONCAT(CONCAT('t', INT_TO_STRING(TsN)), '_avg');
                MessagePackerFb.PackKvLint(ADR(TsKey), DWORD_TO_LINT(TsP^.dwAverageCycleTime));
                TsKey := CONCAT(CONCAT('t', INT_TO_STRING(TsN)), '_max');
                MessagePackerFb.PackKvLint(ADR(TsKey), DWORD_TO_LINT(TsP^.dwMaxCycleTime));
                TsKey := CONCAT(CONCAT('t', INT_TO_STRING(TsN)), '_min');
                MessagePackerFb.PackKvLint(ADR(TsKey), DWORD_TO_LINT(TsP^.dwMinCycleTime));
                TsKey := CONCAT(CONCAT('t', INT_TO_STRING(TsN)), '_jit');
                MessagePackerFb.PackKvDint(ADR(TsKey), TsP^.iJitter);
                TsKey := CONCAT(CONCAT('t', INT_TO_STRING(TsN)), '_jmin');
                MessagePackerFb.PackKvDint(ADR(TsKey), TsP^.iJitterMin);
                TsKey := CONCAT(CONCAT('t', INT_TO_STRING(TsN)), '_jmax');
                MessagePackerFb.PackKvDint(ADR(TsKey), TsP^.iJitterMax);
                TsKey := CONCAT(CONCAT('t', INT_TO_STRING(TsN)), '_cycles');
                MessagePackerFb.PackKvLint(ADR(TsKey), DWORD_TO_LINT(TsP^.dwCycleCount));
                TsKey := CONCAT(CONCAT('t', INT_TO_STRING(TsN)), '_iec_cycles');
                MessagePackerFb.PackKvLint(ADR(TsKey), DWORD_TO_LINT(TsP^.dwIECCycleCount));
                TsN := TsN + 1;
            END_IF;
            IF TsReset THEN
                CmpIecTask.IecTaskResetStatistics(TsH);
            END_IF;
            TsH := CmpIecTask.IecTaskGetNext(ADR('Application'), TsH, ADR(TsR));
        END_WHILE;
        MessagePackerFb.PackKvDint(ADR('n'), TsN);
    ELSIF (CommandType = 'VERSION') THEN
        // Build provenance: lets an external tool verify the running
        // PLC matches a repo commit without IDE assistance. Stamped by
        // codesys_scripts/jobs/stamp_build_info.py before import_all.
        ShouldReturn := TRUE;
        CommandAck := TRUE;
        ResponsePacketPointer^.ele_count := 0;
        MessagePackerFb.PackKvStr(ADR('git_sha'), ADR(GVL.BUILD_GIT_SHA));
        MessagePackerFb.PackKvLint(ADR('build_ts_ms'), GVL.BUILD_TS_MS);
        MessagePackerFb.PackKvLint(ADR('runtime_ms'), AxisGroupSM.RuntimeMs);
    ELSIF (CommandType = 'GET_DIAG') THEN
        // Generic comm/robustness counters dump. UI dashboard polls this
        // (e.g. once per second) to chart drop/NAK/reset rates and the
        // PING gap-jitter envelope. Read-only; doesn't perturb FSM.
        // Counters resettable via SYS/RESET_DBG_INFO (see existing handler).
        ShouldReturn := TRUE;
        CommandAck := TRUE;
        // GET_DIAG fields extended 2026-06-17 to be a TCP-side
        // superset of the daemon-side counter dump the fuzz tests
        // used to call via oapp.read_value. Lets fuzz/soak tests run
        // without the CODESYS RPC daemon being alive -- daemon dies
        // mid-test no longer breaks the test. New fields:
        //   self_reentry, pending_stchg_drop, pending_movedone_drop,
        //   remp_drop_reply, remp_drop_trig, dupe_cmd,
        //   io_cmd_count, io_trig_count, flyevent_avail
        ResponsePacketPointer^.ele_count := 0;
        MessagePackerFb.PackKvDint(ADR('remp_overflow_drop'), TO_DINT(GVL.ReMpOverflowDropCount));
        MessagePackerFb.PackKvLint(ADR('runtime_ms'), AxisGroupSM.RuntimeMs);
        MessagePackerFb.PackKvDint(ADR('sm_scans'), TO_DINT(GVL.AxisGroupSMScans));
        MessagePackerFb.PackKvDint(ADR('remp_drop'), TO_DINT(GVL.ReMpDropCount));
        MessagePackerFb.PackKvDint(ADR('overlen_drop'), TO_DINT(GVL.OverlenDropCount));
        MessagePackerFb.PackKvDint(ADR('send_stall_drop'), TO_DINT(GVL.SendStallDropCount));
        MessagePackerFb.PackKvDint(ADR('group_not_ready_nak'), TO_DINT(GVL.GroupNotReadyNakCount));
        MessagePackerFb.PackKvDint(ADR('missing_type_nak'), TO_DINT(GVL.MissingTypeFieldNakCount));
        MessagePackerFb.PackKvDint(ADR('coord_not_cfg_nak'), TO_DINT(GVL.CoordNotConfiguredNakCount));
        MessagePackerFb.PackKvDint(ADR('proto_mismatch_nak'), TO_DINT(GVL.ProtocolVersionMismatchCount));
        MessagePackerFb.PackKvDint(ADR('idle_reset'), TO_DINT(GVL.IdleResetCount));
        MessagePackerFb.PackKvDint(ADR('read_err_reset'), TO_DINT(GVL.ReadErrorResetCount));
        MessagePackerFb.PackKvDint(ADR('parser_err_reset'), TO_DINT(GVL.ParserErrorResetCount));
        MessagePackerFb.PackKvDint(ADR('write_err_reset'), TO_DINT(GVL.WriteErrorResetCount));
        MessagePackerFb.PackKvDint(ADR('client_connect_count'), TO_DINT(GVL.ClientConnectCount));
        MessagePackerFb.PackKvDint(ADR('server_long_idle_count'), TO_DINT(GVL.ServerLongIdleCount));
        MessagePackerFb.PackKvBool(ADR('server_active'), TCP_MSGPAK_Server.fbMyServer.xServerActive);
        MessagePackerFb.PackKvStr(ADR('bind_addr'), ADR(TCP_MSGPAK_Server.ipServerAddress.ipAddress));
        MessagePackerFb.PackKvDint(ADR('ui_ping_count'), TO_DINT(GVL.UiPingCount));
        MessagePackerFb.PackKvDint(ADR('ui_hb_stale_count'), TO_DINT(GVL.UiHeartbeatStaleCount));
        MessagePackerFb.PackKvDint(ADR('group_error_stop_trips'), TO_DINT(GVL.GroupErrorStopTripCount));
        MessagePackerFb.PackKvDint(ADR('ping_max_gap_ms'), TO_DINT(GVL.PingMaxGapMs));
        MessagePackerFb.PackKvLint(ADR('last_ui_ping_ms'), GVL.LastUiPingMs);
        MessagePackerFb.PackKvDint(ADR('st_chg_event_count'), TO_DINT(GVL.StateChangeEventCount));
        MessagePackerFb.PackKvDint(ADR('self_reentry'), TO_DINT(GVL.SelfReentryCount));
        MessagePackerFb.PackKvDint(ADR('pending_stchg_drop'), TO_DINT(GVL.PendingStChgDropCount));
        MessagePackerFb.PackKvDint(ADR('pending_movedone_drop'), TO_DINT(GVL.PendingMoveDoneDropCount));
        MessagePackerFb.PackKvDint(ADR('remp_drop_reply'), TO_DINT(GVL.ReMpDropCount_Reply));
        MessagePackerFb.PackKvDint(ADR('remp_drop_trig'), TO_DINT(GVL.ReMpDropCount_TriggerEvent));
        MessagePackerFb.PackKvDint(ADR('dupe_cmd'), TO_DINT(GVL.DupeCommandCount));
        // R2/R3/R4/R5/R11: new NAK counters. Published here => they
        // are part of the canonical ResetDiagCounters list (R8).
        MessagePackerFb.PackKvDint(ADR('unknown_cmd_nak'), TO_DINT(GVL.UnknownCmdNakCount));
        MessagePackerFb.PackKvDint(ADR('flyevent_reject_nak'), TO_DINT(GVL.FlyEventRejectNakCount));
        MessagePackerFb.PackKvDint(ADR('flyevent_full_nak'), TO_DINT(GVL.FlyEventBufferFullNakCount));
        MessagePackerFb.PackKvDint(ADR('io_cmd_count'), TO_DINT(AxisGroupSM.IoCommandCount));
        MessagePackerFb.PackKvDint(ADR('io_trig_count'), TO_DINT(AxisGroupSM.IoTriggerCount));
        MessagePackerFb.PackKvDint(ADR('flyevent_avail'), TO_DINT(AxisGroupSM.FlyEventAvailableCount));
ELSE
    CommandAck := FALSE;
    ResponsePacketPointer^.ele_count := 0;
    MessagePackerFb.PackKvStr(ADR('err'), ADR('unknown SYS cmd'));
    UnknownCount := UnknownCount + 1;
END_IF;

MessagePackerFb.PackKvDint(ADR('id'), CommandId);
MessagePackerFb.PackKvBool(ADR('ack'), CommandAck);
IF MsgPakInfoWrapup(DiagInfo) THEN
    OutLen := DiagInfo.buf_size;
    HandledCount := HandledCount + 1;
END_IF;
ReqLen := 0;

(* ---- PRG_EcatEsp.st ---- *)
PROGRAM PRG_EcatEsp
VAR
    byOut0          : USINT;        // bit 0 -> ESP32 LED
    byOut1          : USINT := 16#5A; // echoed back on in1
    byIn0           : USINT;        // ESP32 heartbeat counter
    byIn1           : USINT;        // echo of out1
    byLastIn0       : USINT;
    udiCounterSeen  : UDINT;        // cycles the heartbeat moved
    uiStaleCycles   : UINT;         // cycles since it last moved
    xEspAlive       : BOOL;         // heartbeat moved within 100 cycles
    xRoundTripOk    : BOOL;

    // QY2204-IIC (AS5600) encoder
    uiEncRaw        : UINT;         // 0..4095, one turn
    rEncDeg         : REAL;         // 0..360
    diEncPos        : DINT;         // multi-turn counts, from ESP32 power-up
    rEncTurns       : REAL;         // diEncPos / 4096
    byEncStatus     : USINT;        // bit5 MD, bit4 ML weak, bit3 MH strong, bit0 no sensor
    xMagnetOk       : BOOL;         // MD and neither too weak nor too strong
    xSensorMissing  : BOOL;
    byEncI2cErr     : USINT;
    byEncAgc        : USINT;
END_VAR
(* =========== IMPLEMENTATION =========== *)
GVL.EcProfT1 := LTIME();     // AxisGroupSM done (task timing monitor, PRG_EventLog)
ecat_esp_out0 := byOut0;
ecat_esp_out1 := byOut1;
byIn0 := ecat_esp_in0;
byIn1 := ecat_esp_in1;

IF byIn0 <> byLastIn0 THEN
    udiCounterSeen := udiCounterSeen + 1;
    uiStaleCycles := 0;
ELSIF uiStaleCycles < 65535 THEN
    uiStaleCycles := uiStaleCycles + 1;
END_IF
byLastIn0 := byIn0;
xEspAlive := uiStaleCycles < 100;
xRoundTripOk := (byIn1 = byOut1);

uiEncRaw := USINT_TO_UINT(ecat_esp_in2) OR SHL(USINT_TO_UINT(ecat_esp_in3), 8);
rEncDeg := UINT_TO_REAL(uiEncRaw) * 360.0 / 4096.0;
diEncPos := UDINT_TO_DINT(USINT_TO_UDINT(ecat_esp_in5)
                       OR SHL(USINT_TO_UDINT(ecat_esp_in6), 8)
                       OR SHL(USINT_TO_UDINT(ecat_esp_in7), 16)
                       OR SHL(USINT_TO_UDINT(ecat_esp_in8), 24));
rEncTurns := DINT_TO_REAL(diEncPos) / 4096.0;
byEncStatus := ecat_esp_in4;
xSensorMissing := (byEncStatus AND 16#01) <> 0;
xMagnetOk := ((byEncStatus AND 16#20) <> 0) AND ((byEncStatus AND 16#18) = 0) AND NOT xSensorMissing;
byEncI2cErr := ecat_esp_in9;
byEncAgc := ecat_esp_in10;

(* ---- PRG_EcatEspHttp.st ---- *)
PROGRAM PRG_EcatEspHttp
VAR CONSTANT
    HTML_LEN        : UDINT := 3061;
END_VAR
VAR
    iProfK          : INT;          // Comm task profile
    lrSegUs         : LREAL;
    sHtml           : STRING(3062) := '<!DOCTYPE html><html><head><meta charset="utf-8"><meta name="viewport" content="width=device-width,initial-scale=1"><title>EasyCAT &#32232;&#30908;&#22120;</title><style>body{font-family:system-ui,sans-serif;background:#f4f5f7;color:#1f2328;margin:0;padding:16px}h1{font-size:18px;margin:0 0 12px}.row{display:flex;flex-wrap:wrap;gap:12px}.card{background:#fff;border-radius:10px;padding:14px 16px;box-shadow:0 1px 3px rgba(0,0,0,.08);min-width:150px}.k{font-size:12px;color:#656d76}.v{font-size:26px;font-weight:600;font-variant-numeric:tabular-nums}.ok{color:#1a7f37}.bad{color:#cf222e}.warn{color:#9a6700}svg{display:block}#conn{font-size:12px;color:#656d76;margin-top:12px}</style></head><body><h1>EasyCAT + ESP32 &#32232;&#30908;&#22120;&#29376;&#24907;</h1><div class="row"><div class="card"><svg width="170" height="170" viewBox="-85 -85 170 170"><circle r="78" fill="#f4f5f7" stroke="#d0d7de" stroke-width="2"/><line id="nd" x1="0" y1="0" x2="0" y2="-68" stroke="#0969da" stroke-width="5" stroke-linecap="round"/><circle r="5" fill="#0969da"/></svg></div><div class="card"><div class="k">&#35282;&#24230;</div><div class="v" id="deg">-</div><div class="k" style="margin-top:10px">&#21407;&#22987;&#20540; (0-4095)</div><div class="v" id="raw">-</div></div><div class="card"><div class="k">&#22810;&#22280;&#20301;&#32622; (counts)</div><div class="v" id="pos">-</div><div class="k" style="margin-top:10px">&#22280;&#25976;</div><div class="v" id="turns">-</div></div></div><div class="row" style="margin-top:12px"><div class="card"><div class="k">ESP32</div><div class="v" id="alive">-</div></div><div class="card"><div class="k">EtherCAT</div><div class="v" id="ecat">-</div></div><div class="card"><div class="k">&#30913;&#37941;</div><div class="v" id="mag">-</div></div><div class="card"><div class="k">AGC / I2C &#37679;&#35492;</div><div class="v" id="agc">-</div></div></div><div id="conn">-</div><script>var S={1:"INIT",2:"PREOP",3:"BOOT",4:"SAFEOP",8:"OP"};function g(i){return document.getElementById(i)}function put(i,h,c){var e=g(i);e.innerHTML=h;e.className="v "+(c||"")}function tick(){fetch("/s",{cache:"no-store"}).then(function(r){return r.json()}).then(function(j){var deg=j.raw*360/4096;g("nd").setAttribute("transform","rotate("+deg.toFixed(1)+")");put("deg",deg.toFixed(1)+"&deg;");put("raw",j.raw);put("pos",j.pos);put("turns",(j.pos/4096).toFixed(3));put("alive",j.alive?"&#36939;&#20316;&#20013;":"&#28961;&#24515;&#36339;",j.alive?"ok":"bad");put("ecat",S[j.ecat]||j.ecat,j.ecat==8?"ok":"bad");var m=j.st&1?["&#28961;&#24863;&#28204;&#22120;","bad"]:j.st&16?["&#22826;&#24369;","warn"]:j.st&8?["&#22826;&#24375;","warn"]:j.st&32?["&#27491;&#24120;","ok"]:["&#26410;&#20597;&#28204;","bad"];put("mag",m[0],m[1]);put("agc",j.agc+" / "+j.err);g("conn").innerHTML="&#26356;&#26032; "+new Date().toLocaleTimeString()+" &middot; &#35531;&#27714; "+j.hb;setTimeout(tick,200)}).catch(function(){g("conn").innerHTML="&#36899;&#32218;&#20013;&#26039;&#65292;&#37325;&#35430;&#20013;";setTimeout(tick,1000)})}tick();</script></body></html>';
    sHdrHtml        : STRING(200) := 'HTTP/1.1 200 OK$R$NContent-Type: text/html; charset=utf-8$R$NCache-Control: no-store$R$NConnection: close$R$N$R$N';
    sHdrJson        : STRING(200) := 'HTTP/1.1 200 OK$R$NContent-Type: application/json$R$NCache-Control: no-store$R$NConnection: close$R$N$R$N';
    sHdrText        : STRING(200) := 'HTTP/1.1 200 OK$R$NContent-Type: text/plain$R$NCache-Control: no-store$R$NConnection: close$R$N$R$N';
    sHdr404         : STRING(120) := 'HTTP/1.1 404 Not Found$R$NContent-Length: 0$R$NConnection: close$R$N$R$N';
    sJson           : STRING(255);

    ipAny           : NBS.IPv4Address := (ipAddress:='0.0.0.0');
    fbServer        : NBS.TCP_Server := (itfIPAddress:=ipAny, uiPort:=8126, xEnable:=TRUE, udiMaxConnections:=1);
    fbConn          : NBS.TCP_Connection;
    itfServer       : NBS.IServer;

    abyReq          : ARRAY[0..511] OF BYTE;
    udiReqCount     : UDINT;
    eRx             : NBS.ERROR;
    eTx             : NBS.ERROR;
    xReset          : BOOL;
    xResponded      : BOOL;
    uiCloseDelay    : UINT;
    udiRequests     : UDINT;
    // GET /e?s=<seq>: event log (GVL.EvHead) from <seq>, text lines
    // "seq t_ms kind val", first line "head <EvHead>". At most EV_MAX
    // lines per request; the client asks again from the last seq + 1.
    abyEv           : ARRAY[0..6143] OF BYTE;
    udiEvLen        : UDINT;
    udiEvFrom       : UDINT;
    udiEvTo         : UDINT;
    udiEvHead       : UDINT;
    udiEvSeq        : UDINT;
    udiEvSlot       : UDINT;
    iEvPos          : INT;
    sEvLine         : STRING(60);
    EV_MAX          : UDINT := 150;
    // One connection at a time: a client that connects and never sends a
    // request (killed mid-request) held it forever and every later request
    // was refused (seen 2026-09-24). Drop it after 1 s.
    tonIdle         : TON;
    udiIdleDrops    : UDINT;
    // Also seen: after a client vanished the connection FB sat enabled but
    // neither busy nor active -- no error, never listening again. Re-arm
    // it after a few such scans (debounced: xBusy may lag the enable).
    uiDeadScans     : UINT;
    udiRearms       : UDINT;

    // ---- Stream on :8128: one persistent connection, the PLC pushes lines
    // (no request, no reconnect per sample -- the HTTP polling above costs
    // a connect/close per request and stalls when a SYN is dropped).
    //   e <seq> <t_ms> <kind> <val>      every GVL.EvHead event, from connect time
    //   v <sd> <bt> <ff> <tp> <ad> <rp> <bx> <by>   PRG_SimIo counters, every 20 ms
    // Used by tools/sim/vision_mock.py.
    fbStreamSrv     : NBS.TCP_Server := (itfIPAddress:=ipAny, uiPort:=8128, xEnable:=TRUE, udiMaxConnections:=1);
    fbStream        : NBS.TCP_Connection;
    xStreamReset    : BOOL;
    xStreamOn       : BOOL;
    uiStreamDead    : UINT;
    udiStreamSeq    : UDINT;
    udiStreamHead   : UDINT;
    udiStreamSlot   : UDINT;
    udiStreamLen    : UDINT;
    iStreamLines    : INT;
    lStreamLastV    : LINT;
    sStreamLine     : STRING(120);
    abyStream       : ARRAY[0..4095] OF BYTE;
    eStreamTx       : NBS.ERROR;
    udiStreamClients : UDINT;
    udiStreamLost   : UDINT;
    udiStreamWriteErr : UDINT;
END_VAR
(* =========== IMPLEMENTATION =========== *)
GVL.CommT[2] := LTIME(); GVL.CommCyc[2] := GVL.EcProfCycles;   // Comm task profile
fbServer();
itfServer := fbServer.itfServer;
fbConn(itfServer := itfServer, xEnable := (itfServer <> 0) AND NOT xReset);
// A reset is complete once the FB has been called disabled and is idle;
// the next scan enables it again (a clean enable edge).
IF xReset AND NOT fbConn.xActive AND NOT fbConn.xBusy THEN
    xReset := FALSE;
    xResponded := FALSE;
    uiDeadScans := 0;
END_IF
IF (itfServer <> 0) AND NOT xReset AND NOT fbConn.xBusy AND NOT fbConn.xActive THEN
    uiDeadScans := uiDeadScans + 1;
    IF uiDeadScans > 10 THEN
        udiRearms := udiRearms + 1;
        xReset := TRUE;
    END_IF
ELSE
    uiDeadScans := 0;
END_IF

IF fbConn.xActive AND NOT xResponded THEN
    eRx := fbConn.Read(ADR(abyReq), SIZEOF(abyReq), udiCount => udiReqCount);
    IF eRx = NBS.ERROR.NO_ERROR AND udiReqCount >= 6 THEN
        udiRequests := udiRequests + 1;
        // Request line: "GET /s" -> status JSON, "GET /v" -> sim JSON,
        // "GET / " -> page.
        IF abyReq[5] = 16#73 THEN
            sJson := '{"alive":';
            IF PRG_EcatEsp.xEspAlive THEN sJson := CONCAT(sJson, '1'); ELSE sJson := CONCAT(sJson, '0'); END_IF
            sJson := CONCAT(sJson, ',"ecat":');
            sJson := CONCAT(sJson, UINT_TO_STRING(TO_UINT(EasyCAT.wState)));
            sJson := CONCAT(sJson, ',"raw":');
            sJson := CONCAT(sJson, UINT_TO_STRING(PRG_EcatEsp.uiEncRaw));
            sJson := CONCAT(sJson, ',"pos":');
            sJson := CONCAT(sJson, DINT_TO_STRING(PRG_EcatEsp.diEncPos));
            sJson := CONCAT(sJson, ',"st":');
            sJson := CONCAT(sJson, USINT_TO_STRING(PRG_EcatEsp.byEncStatus));
            sJson := CONCAT(sJson, ',"err":');
            sJson := CONCAT(sJson, USINT_TO_STRING(PRG_EcatEsp.byEncI2cErr));
            sJson := CONCAT(sJson, ',"agc":');
            sJson := CONCAT(sJson, USINT_TO_STRING(PRG_EcatEsp.byEncAgc));
            sJson := CONCAT(sJson, ',"hb":');
            sJson := CONCAT(sJson, UDINT_TO_STRING(udiRequests));
            sJson := CONCAT(sJson, '}');
            eTx := fbConn.Write(ADR(sHdrJson), INT_TO_UDINT(LEN(sHdrJson)));
            eTx := fbConn.Write(ADR(sJson), INT_TO_UDINT(LEN(sJson)));
        ELSIF abyReq[5] = 16#76 THEN
            sJson := '{"sd":';
            sJson := CONCAT(sJson, UDINT_TO_STRING(PRG_SimIo.udiSide));
            sJson := CONCAT(sJson, ',"bt":');
            sJson := CONCAT(sJson, UDINT_TO_STRING(PRG_SimIo.udiBtm));
            sJson := CONCAT(sJson, ',"ff":');
            sJson := CONCAT(sJson, UDINT_TO_STRING(PRG_SimIo.udiFeeder));
            sJson := CONCAT(sJson, ',"tp":');
            sJson := CONCAT(sJson, UDINT_TO_STRING(PRG_SimIo.udiTop));
            sJson := CONCAT(sJson, ',"ad":');
            sJson := CONCAT(sJson, UDINT_TO_STRING(PRG_SimIo.udiReelAdv));
            sJson := CONCAT(sJson, ',"rp":');
            sJson := CONCAT(sJson, LREAL_TO_STRING(reelpullmotor.fActPosition));
            sJson := CONCAT(sJson, ',"bx":');
            sJson := CONCAT(sJson, REAL_TO_STRING(PRG_SimIo.rBtmX));
            sJson := CONCAT(sJson, ',"by":');
            sJson := CONCAT(sJson, REAL_TO_STRING(PRG_SimIo.rBtmY));
            sJson := CONCAT(sJson, '}');
            eTx := fbConn.Write(ADR(sHdrJson), INT_TO_UDINT(LEN(sHdrJson)));
            eTx := fbConn.Write(ADR(sJson), INT_TO_UDINT(LEN(sJson)));
        ELSIF abyReq[5] = 16#65 THEN
            // "GET /e?s=123 ..." -- parse the digits after "?s=".
            udiEvFrom := 0;
            IF abyReq[6] = 16#3F AND abyReq[7] = 16#73 AND abyReq[8] = 16#3D THEN
                iEvPos := 9;
                WHILE (iEvPos < 40) AND (abyReq[iEvPos] >= 16#30) AND (abyReq[iEvPos] <= 16#39) DO
                    udiEvFrom := udiEvFrom * 10 + BYTE_TO_UDINT(abyReq[iEvPos] - 16#30);
                    iEvPos := iEvPos + 1;
                END_WHILE
            END_IF
            udiEvHead := GVL.EvHead;
            // Keep clear of slots the writer may be reusing.
            IF (udiEvHead > 1000) AND (udiEvFrom < udiEvHead - 1000) THEN
                udiEvFrom := udiEvHead - 1000;
            END_IF
            udiEvTo := udiEvHead;
            IF (udiEvTo > udiEvFrom + EV_MAX) THEN udiEvTo := udiEvFrom + EV_MAX; END_IF
            sEvLine := CONCAT('head ', UDINT_TO_STRING(udiEvHead));
            sEvLine := CONCAT(sEvLine, '$N');
            udiEvLen := INT_TO_UDINT(LEN(sEvLine));
            MEMUtils.MemCpy(ADR(abyEv[0]), ADR(sEvLine), INT_TO_UINT(LEN(sEvLine)));
            udiEvSeq := udiEvFrom;
            WHILE udiEvSeq < udiEvTo DO
                udiEvSlot := udiEvSeq MOD 1024;
                sEvLine := CONCAT(UDINT_TO_STRING(udiEvSeq), ' ');
                sEvLine := CONCAT(sEvLine, UDINT_TO_STRING(GVL.EvT[udiEvSlot]));
                sEvLine := CONCAT(sEvLine, ' ');
                sEvLine := CONCAT(sEvLine, BYTE_TO_STRING(GVL.EvKind[udiEvSlot]));
                sEvLine := CONCAT(sEvLine, ' ');
                sEvLine := CONCAT(sEvLine, UDINT_TO_STRING(GVL.EvVal[udiEvSlot]));
                sEvLine := CONCAT(sEvLine, '$N');
                MEMUtils.MemCpy(ADR(abyEv[udiEvLen]), ADR(sEvLine), INT_TO_UINT(LEN(sEvLine)));
                udiEvLen := udiEvLen + INT_TO_UDINT(LEN(sEvLine));
                udiEvSeq := udiEvSeq + 1;
            END_WHILE
            eTx := fbConn.Write(ADR(sHdrText), INT_TO_UDINT(LEN(sHdrText)));
            eTx := fbConn.Write(ADR(abyEv), udiEvLen);
        ELSIF abyReq[5] = 16#20 THEN
            eTx := fbConn.Write(ADR(sHdrHtml), INT_TO_UDINT(LEN(sHdrHtml)));
            eTx := fbConn.Write(ADR(sHtml), HTML_LEN);
        ELSE
            eTx := fbConn.Write(ADR(sHdr404), INT_TO_UDINT(LEN(sHdr404)));
        END_IF
        xResponded := TRUE;
        uiCloseDelay := 0;
    END_IF
END_IF

tonIdle(IN := fbConn.xActive AND NOT xResponded, PT := T#1S);
IF tonIdle.Q THEN
    udiIdleDrops := udiIdleDrops + 1;
    xReset := TRUE;
END_IF

// Give the stack a few cycles to flush, then close ("Connection: close").
IF xResponded THEN
    uiCloseDelay := uiCloseDelay + 1;
    IF uiCloseDelay > 5 THEN
        xReset := TRUE;
    END_IF
END_IF
IF fbConn.xError THEN
    xReset := TRUE;
END_IF

// ---- Event / counter stream on :8128 -------------------------------------
fbStreamSrv();
fbStream(itfServer := fbStreamSrv.itfServer, xEnable := (fbStreamSrv.itfServer <> 0) AND NOT xStreamReset);
IF xStreamReset AND NOT fbStream.xActive AND NOT fbStream.xBusy THEN
    xStreamReset := FALSE;
    xStreamOn := FALSE;
    uiStreamDead := 0;
END_IF
// Same re-arm as the HTTP connection: enabled but neither busy nor active.
IF (fbStreamSrv.itfServer <> 0) AND NOT xStreamReset AND NOT fbStream.xBusy AND NOT fbStream.xActive THEN
    uiStreamDead := uiStreamDead + 1;
    IF uiStreamDead > 10 THEN
        xStreamReset := TRUE;
    END_IF
ELSE
    uiStreamDead := 0;
END_IF

IF fbStream.xActive AND NOT xStreamReset THEN
    IF NOT xStreamOn THEN
        xStreamOn := TRUE;
        udiStreamSeq := GVL.EvHead;          // from now on
        lStreamLastV := 0;
        udiStreamClients := udiStreamClients + 1;
    END_IF
    udiStreamLen := 0;
    udiStreamHead := GVL.EvHead;
    IF (udiStreamHead > 1000) AND (udiStreamSeq < udiStreamHead - 1000) THEN
        udiStreamLost := udiStreamLost + (udiStreamHead - 1000 - udiStreamSeq);
        udiStreamSeq := udiStreamHead - 1000;
    END_IF
    iStreamLines := 0;
    WHILE (udiStreamSeq < udiStreamHead) AND (iStreamLines < 60) DO
        udiStreamSlot := udiStreamSeq MOD 1024;
        sStreamLine := CONCAT('e ', UDINT_TO_STRING(udiStreamSeq));
        sStreamLine := CONCAT(sStreamLine, ' ');
        sStreamLine := CONCAT(sStreamLine, UDINT_TO_STRING(GVL.EvT[udiStreamSlot]));
        sStreamLine := CONCAT(sStreamLine, ' ');
        sStreamLine := CONCAT(sStreamLine, BYTE_TO_STRING(GVL.EvKind[udiStreamSlot]));
        sStreamLine := CONCAT(sStreamLine, ' ');
        sStreamLine := CONCAT(sStreamLine, UDINT_TO_STRING(GVL.EvVal[udiStreamSlot]));
        sStreamLine := CONCAT(sStreamLine, '$N');
        MEMUtils.MemCpy(ADR(abyStream[udiStreamLen]), ADR(sStreamLine), INT_TO_UINT(LEN(sStreamLine)));
        udiStreamLen := udiStreamLen + INT_TO_UDINT(LEN(sStreamLine));
        udiStreamSeq := udiStreamSeq + 1;
        iStreamLines := iStreamLines + 1;
    END_WHILE
    IF (AxisGroupSM.RuntimeMs - lStreamLastV) >= 20 THEN
        lStreamLastV := AxisGroupSM.RuntimeMs;
        sStreamLine := CONCAT('v ', UDINT_TO_STRING(PRG_SimIo.udiSide));
        sStreamLine := CONCAT(sStreamLine, ' ');
        sStreamLine := CONCAT(sStreamLine, UDINT_TO_STRING(PRG_SimIo.udiBtm));
        sStreamLine := CONCAT(sStreamLine, ' ');
        sStreamLine := CONCAT(sStreamLine, UDINT_TO_STRING(PRG_SimIo.udiFeeder));
        sStreamLine := CONCAT(sStreamLine, ' ');
        sStreamLine := CONCAT(sStreamLine, UDINT_TO_STRING(PRG_SimIo.udiTop));
        sStreamLine := CONCAT(sStreamLine, ' ');
        sStreamLine := CONCAT(sStreamLine, UDINT_TO_STRING(PRG_SimIo.udiReelAdv));
        sStreamLine := CONCAT(sStreamLine, ' ');
        sStreamLine := CONCAT(sStreamLine, LREAL_TO_STRING(reelpullmotor.fActPosition));
        sStreamLine := CONCAT(sStreamLine, ' ');
        sStreamLine := CONCAT(sStreamLine, REAL_TO_STRING(PRG_SimIo.rBtmX));
        sStreamLine := CONCAT(sStreamLine, ' ');
        sStreamLine := CONCAT(sStreamLine, REAL_TO_STRING(PRG_SimIo.rBtmY));
        sStreamLine := CONCAT(sStreamLine, '$N');
        MEMUtils.MemCpy(ADR(abyStream[udiStreamLen]), ADR(sStreamLine), INT_TO_UINT(LEN(sStreamLine)));
        udiStreamLen := udiStreamLen + INT_TO_UDINT(LEN(sStreamLine));
    END_IF
    IF udiStreamLen > 0 THEN
        eStreamTx := fbStream.Write(ADR(abyStream), udiStreamLen);
        IF eStreamTx <> NBS.ERROR.NO_ERROR THEN
            // client gone or send buffer full: drop it, it reconnects
            udiStreamWriteErr := udiStreamWriteErr + 1;
            xStreamReset := TRUE;
        END_IF
    END_IF
END_IF
IF fbStream.xError THEN
    xStreamReset := TRUE;
END_IF

// ---- Comm task profile (GVL.Comm*): the last POU of the Comm task ----
GVL.CommT[3] := LTIME();
GVL.CommCyc[3] := GVL.EcProfCycles;
IF GVL.CommProfReset THEN
    GVL.CommProfReset := FALSE;
    FOR iProfK := 0 TO 2 DO
        GVL.CommSegUsMax[iProfK] := 0;
        GVL.CommSegBusCyc[iProfK] := 0;
        GVL.CommSegOver1ms[iProfK] := 0;
    END_FOR;
    GVL.CommScanUsMax := 0;
    GVL.CommOutsideUsMax := 0;
    GVL.CommTaskUsMax := 0;
    GVL.CommOutsideOver500 := 0;
END_IF;
FOR iProfK := 0 TO 2 DO
    lrSegUs := ULINT_TO_LREAL(LTIME_TO_ULINT(GVL.CommT[iProfK + 1] - GVL.CommT[iProfK])) / 1000.0;
    IF lrSegUs > GVL.CommSegUsMax[iProfK] THEN
        GVL.CommSegUsMax[iProfK] := lrSegUs;
        GVL.CommSegBusCyc[iProfK] := GVL.CommCyc[iProfK + 1] - GVL.CommCyc[iProfK];
    END_IF;
    IF lrSegUs > 1000.0 THEN
        GVL.CommSegOver1ms[iProfK] := GVL.CommSegOver1ms[iProfK] + 1;
    END_IF;
END_FOR;
GVL.CommScanUsLast := ULINT_TO_LREAL(LTIME_TO_ULINT(GVL.CommT[3] - GVL.CommT[0])) / 1000.0;
GVL.CommScanUsMax := MAX(GVL.CommScanUsMax, GVL.CommScanUsLast);

(* ---- PRG_EcatStepper.st ---- *)
PROGRAM PRG_EcatStepper
VAR CONSTANT
    CYCLE_S             : LREAL := 0.001;   // EtherCAT_Task cycle, s (DT is a keyword)
    MAX_STEPS_PER_CYCLE : LREAL := 135.0;   // firmware faults above 150
END_VAR
VAR
    // --- interface ---
    xEnable         : BOOL;
    rTargetDeg      : LREAL;
    rMaxVelDeg      : LREAL := 180.0;       // deg/s
    rAccDeg         : LREAL := 1800.0;      // deg/s^2
    udiStepsPerRev  : UDINT := 6400;        // 200 full steps x 32 microsteps
    xSetZero        : BOOL;
    xReset          : BOOL;

    rActualDeg      : LREAL;
    rCmdDeg         : LREAL;
    xInPosition     : BOOL;
    xEnabled        : BOOL;
    xFault          : BOOL;
    byFault         : USINT;                // 1 comm lost, 2 setpoint jump

    // --- internals ---
    diActual        : DINT;                 // steps emitted, from the ESP32
    diCmd           : DINT;                 // setpoint sent this cycle
    diZero          : DINT;
    lrPos           : LREAL;                // profile position, steps
    lrVel           : LREAL;                // profile velocity, steps/s
    lrTarget        : LREAL;
    lrErr           : LREAL;
    lrVmax          : LREAL;
    lrAcc           : LREAL;
    lrVdes          : LREAL;
    lrStep          : LREAL;
    lrScale         : LREAL;                // steps per degree
    xActive         : BOOL;
    xLastSetZero    : BOOL;
    udiCmd          : UDINT;
END_VAR
(* =========== IMPLEMENTATION =========== *)
diActual := UDINT_TO_DINT(USINT_TO_UDINT(ecat_esp_in16)
                       OR SHL(USINT_TO_UDINT(ecat_esp_in17), 8)
                       OR SHL(USINT_TO_UDINT(ecat_esp_in18), 16)
                       OR SHL(USINT_TO_UDINT(ecat_esp_in19), 24));
xEnabled := (ecat_esp_in20 AND 16#01) <> 0;
xFault := (ecat_esp_in20 AND 16#02) <> 0;
byFault := ecat_esp_in21;

lrScale := UDINT_TO_LREAL(MAX(udiStepsPerRev, 1)) / 360.0;

// Zero at the current position; hold still there.
IF xSetZero AND NOT xLastSetZero THEN
    diZero := diActual;
    rTargetDeg := 0.0;
    lrPos := DINT_TO_LREAL(diActual);
    lrVel := 0.0;
END_IF
xLastSetZero := xSetZero;

rActualDeg := DINT_TO_LREAL(diActual - diZero) / lrScale;
lrTarget := DINT_TO_LREAL(diZero) + rTargetDeg * lrScale;

IF xEnable AND NOT xFault THEN
    IF NOT xActive THEN
        // Start from where the motor is, so the first setpoint is no jump.
        lrPos := DINT_TO_LREAL(diActual);
        lrVel := 0.0;
        xActive := TRUE;
    END_IF

    lrVmax := MIN(ABS(rMaxVelDeg) * lrScale, MAX_STEPS_PER_CYCLE / CYCLE_S);
    lrAcc := MAX(ABS(rAccDeg) * lrScale, 1.0);
    lrErr := lrTarget - lrPos;

    // Velocity that still stops exactly at the target: sqrt(2 a |e|),
    // capped at vmax; approach it at most a*dt per cycle.
    lrVdes := MIN(lrVmax, SQRT(2.0 * lrAcc * ABS(lrErr)));
    IF lrErr < 0.0 THEN
        lrVdes := -lrVdes;
    END_IF
    IF lrVdes > lrVel + lrAcc * CYCLE_S THEN
        lrVel := lrVel + lrAcc * CYCLE_S;
    ELSIF lrVdes < lrVel - lrAcc * CYCLE_S THEN
        lrVel := lrVel - lrAcc * CYCLE_S;
    ELSE
        lrVel := lrVdes;
    END_IF

    lrStep := lrVel * CYCLE_S;
    IF (lrErr >= 0.0 AND lrStep > lrErr) OR (lrErr <= 0.0 AND lrStep < lrErr) THEN
        lrStep := lrErr;                    // land on the target, no overshoot
        lrVel := 0.0;
    END_IF
    lrPos := lrPos + lrStep;
    diCmd := LREAL_TO_DINT(lrPos);
    ecat_esp_out2 := 16#01;                 // enable
ELSE
    // Disabled or faulted: follow the motor, send no motion.
    xActive := FALSE;
    lrVel := 0.0;
    lrPos := DINT_TO_LREAL(diActual);
    diCmd := diActual;
    IF xReset THEN
        ecat_esp_out2 := 16#02;             // fault reset, enable off
    ELSE
        ecat_esp_out2 := 16#00;
    END_IF
END_IF

rCmdDeg := (lrPos - DINT_TO_LREAL(diZero)) / lrScale;
xInPosition := xEnabled AND lrVel = 0.0 AND ABS(lrTarget - DINT_TO_LREAL(diActual)) < 1.0;

udiCmd := DINT_TO_UDINT(diCmd);
ecat_esp_out4 := UDINT_TO_USINT(udiCmd AND 16#FF);
ecat_esp_out5 := UDINT_TO_USINT(SHR(udiCmd, 8) AND 16#FF);
ecat_esp_out6 := UDINT_TO_USINT(SHR(udiCmd, 16) AND 16#FF);
ecat_esp_out7 := UDINT_TO_USINT(SHR(udiCmd, 24) AND 16#FF);
